RoboDK station: kr30 cnc 040719 4.rdk

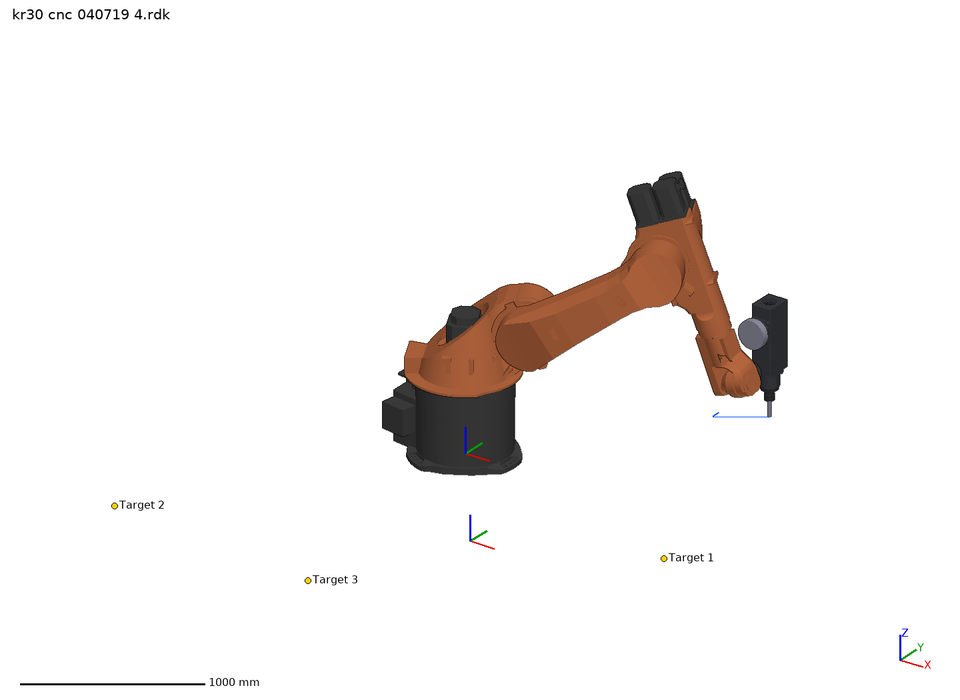
[picture v0: the station drawn from its stored meshes, robots at their saved joint values, targets as dots, program paths as lines]
Station kr30 cnc 040719 4. Poses are relative to the parent item; angles as X-Y-Z fixed-axis rotations.
  - frame KUKA KR 30 HA Base at (0, 0, 0) mm
    - robot KUKA KR 30 HA: 6 axes, payload 30 kg, reach 2033 mm, repeatability 0.05 mm, weight 665 kg
        modified DH rows (alpha deg, a mm, theta deg, d mm): 0, 0, 0, 815; -90, 350, 0, 0; 0, 850, -90, 0; -90, 145, 0, 820; 90, 0, 0, 0; -90, 0, 180, 170
        joint limits [-185, -135, -120, -350, -119, -350] to [185, 35, 158, 350, 119, 350]; home [0, -90, 90, 0, 0, 0]; saved at [-26.942, -31.651, 103.522, 244.219, 81.895, -196.272]
      - tool 1/2" End Mill TCP, TCP at (337.71, -2.2, 160.57) mm, size 692.9 x 170 x 256 mm
    - frame Reference Rhino at (865.96, -1191.99, 189.15) mm
      - target Target 1 (Cartesian target) at (994.45, 406.4, 10) mm, rotated rx 0 ry 90 rz -60.43 deg; joints [10.582, -19.112, 71.071, -56.398, -66.586, 30.882] of KUKA KR 30 HA
      - target Target 2 (Cartesian target) at (-1810.84, -765.32, 10.08) mm, rotated rx 49.23 ry 89.99 rz -110.09 deg; joints [109.49, -19.11, 71.06, -56.39, -66.58, 30.88] of KUKA KR 30 HA
      - target Target 3 (Cartesian target) at (-425.52, -920.6, 10.08) mm, rotated rx 49.23 ry 89.99 rz -69.31 deg; joints [68.71, -19.11, 71.06, -56.39, -66.58, 30.88] of KUKA KR 30 HA
      - object RhinoPart at (0, 0, 0) mm
  - machining project RhinoPart Settings: C:/Users/Julian Ramirez.DESKTOP-JVDE542/Desktop/ELMER SHEET 1 TEST 3.nc | rotZ(0) | rotX(00)*rotY(360) | rotZ(0)*rotY(270)
  - object box at (500, 500, 500) mm, size 250 x 250 x 250 mm, geometry from box.sld
  - program RhinoPart (11 instructions, listed below)
  - program Prog2 (1 instructions, listed below)
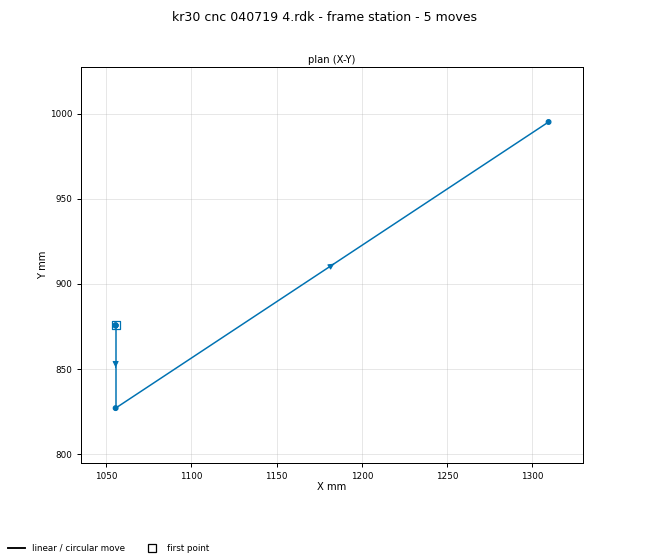
[picture p0: tool path of kr30 cnc 040719 4.rdk in frame station, 5 of 6 moves have a stored position in this frame; points joined in program order, loops and branches not executed]

--- program RhinoPart (robot KUKA KR 30 HA) ---
  Smooth(1)
  Set Ref.: Reference Rhino
  Set Tool: 1/2" End Mill TCP
  Show 1/2" End Mill TCP
  Set speed (2000.0 mm/s)
  MoveJ 1 to (189.6, 2067.69, 0) mm, rotated rx 0 ry 90 rz -90 deg; joints [-48.753, -26.677, 90.247, 44.399, 109.552, -161.855]
  MoveL 2 to (189.6, 2067.69, 0) mm, rotated rx 0 ry 90 rz -90 deg; joints [-48.753, -26.677, 90.247, 44.399, 109.552, -161.855]
  MoveL 3 to (189.6, 2067.69, 0) mm, rotated rx 0 ry 90 rz -90 deg; joints [-48.753, -26.677, 90.247, 44.399, 109.552, -161.855]
  Set speed (60.0 mm/s)
  MoveL 4 to (189.6, 2019.15, 0) mm, rotated rx 0 ry 90 rz 33.46 deg; joints [-39.715, -39.838, 139.216, 173.662, 99.321, -181.031]
  MoveL 5 to (443.6, 2187.03, 0) mm, rotated rx 0 ry 90 rz 90 deg; joints [-26.942, -31.651, 103.522, 244.219, 81.895, -196.272]

--- program Prog2 (robot KUKA KR 30 HA) ---
  MoveC [its target is no longer in the station] [its target is no longer in the station]
